SUBAPPLICATION MessageExchangeDemo (* SoA implementation in function blocks (slide 47): WorkpieceSensor -> CylinderOrchestrator -> CylinderService / DropSinkService, coupled via three EVENT_HS_WSTRING-family adapter connections *)
  (* Standard: 61499-2; Description: Copyright (c) 2026 Meisterschulen am Ostbahnhof This program and the accompanying materials are made available under the terms of the Eclipse Public License 2.0 which is available at https://www.eclipse.org/legal/epl-2.0/ SPDX-License-Identifier: EPL-2.0 *)
  (* Version 1.0, 2026-09-03, Franz Höpfinger, Meisterschulen am Ostbahnhof, SoA implementation in function blocks (IEC 61499 primer course, Module 6, Valeriy Vyatkin, slide 47), demo application reconstructing the CylH message exchange (slides 42-46) as four cooperating function blocks *)
  PACKAGE Meins::DesingPatterns::HandshakePattern;
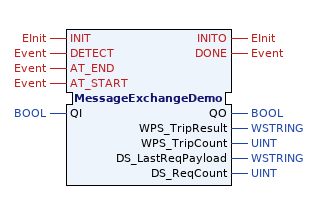
  EVENT_INPUT
    INIT : EInit; (* Initialization Request *)
    DETECT; (* Simulated WPS sensor: a workpiece has arrived, starts the round trip *)
    AT_END; (* Simulated CYL.end sensor: pusher reached the end position *)
    AT_START; (* Simulated CYL.start sensor: pusher reached the start position again *)
  END_EVENT
  EVENT_OUTPUT
    INITO : EInit; (* Initialization Confirm *)
    DONE; (* WorkpieceSensor received the CNF confirming the round trip is complete *)
  END_EVENT
  VAR_INPUT
    QI : BOOL; (* Input event qualifier *)
  END_VAR
  VAR_OUTPUT
    QO : BOOL; (* Output event qualifier *)
    WPS_TripResult : WSTRING; (* WorkpieceSensor: payload of the last received CNF (expect RSP_CYL_TRIP_COMPLETE) *)
    WPS_TripCount : UINT; (* WorkpieceSensor: number of completed round trips *)
    DS_LastReqPayload : WSTRING; (* DropSinkService: payload of the last received REQ (expect REQ_DROP) *)
    DS_ReqCount : UINT; (* DropSinkService: number of drop REQ received *)
  END_VAR
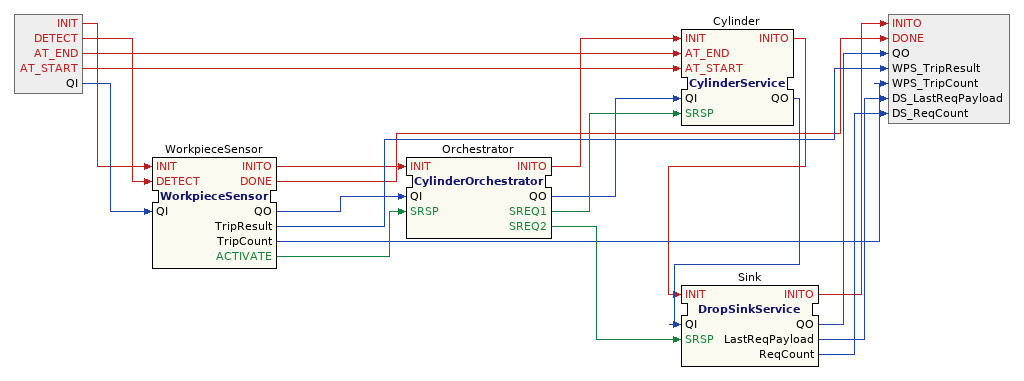
  FBS
    WorkpieceSensor : Meins::DesingPatterns::HandshakePattern::WorkpieceSensor;
    Orchestrator : Meins::DesingPatterns::HandshakePattern::CylinderOrchestrator;
    Cylinder : Meins::DesingPatterns::HandshakePattern::CylinderService;
    Sink : Meins::DesingPatterns::HandshakePattern::DropSinkService;
  END_FBS
  EVENT_CONNECTIONS
    INIT TO WorkpieceSensor.INIT;
    WorkpieceSensor.INITO TO Orchestrator.INIT;
    Orchestrator.INITO TO Cylinder.INIT;
    Cylinder.INITO TO Sink.INIT;
    Sink.INITO TO INITO;
    DETECT TO WorkpieceSensor.DETECT;
    AT_END TO Cylinder.AT_END;
    AT_START TO Cylinder.AT_START;
    WorkpieceSensor.DONE TO DONE;
  END_CONNECTIONS
  DATA_CONNECTIONS
    QI TO WorkpieceSensor.QI;
    WorkpieceSensor.QO TO Orchestrator.QI;
    Orchestrator.QO TO Cylinder.QI;
    Cylinder.QO TO Sink.QI;
    Sink.QO TO QO;
    WorkpieceSensor.TripResult TO WPS_TripResult;
    WorkpieceSensor.TripCount TO WPS_TripCount;
    Sink.LastReqPayload TO DS_LastReqPayload;
    Sink.ReqCount TO DS_ReqCount;
  END_CONNECTIONS
  ADAPTER_CONNECTIONS
    WorkpieceSensor.ACTIVATE TO Orchestrator.SRSP; (* WorkpieceSensor requests the round trip (REQ_TRIP); Orchestrator answers once the whole trip is confirmed complete *)
    Orchestrator.SREQ1 TO Cylinder.SRSP; (* Orchestrator forwards the trip request; reacts to the mid-trip IND (end position reached) and the closing CNF (trip complete) *)
    Orchestrator.SREQ2 TO Sink.SRSP; (* Orchestrator requests the drop once the cylinder reports reaching the end position *)
  END_CONNECTIONS
END_SUBAPPLICATION
